Fanuc KAREL source: kt00483.KL

-- PROVISIONAL review KL for V770-1; original PC SHA256 eedee7176f4b0b8d41bb8e5626b35325a9c50e701c9c6c733b56d75d0fa50af2
-- Incomplete behavior may be omitted. Consult companion uncertainty JSON. Do not deploy.
PROGRAM KT00483
%NOLOCKGROUP
VAR
  OUT : BOOLEAN
-- UNRESOLVED_DECL P1 type=000101
-- UNRESOLVED_DECL P2 type=000106
BEGIN
  -- UNRESOLVED_PC offsets 5-20; opcodes 2E,22,32,35
  -- UNRESOLVED_PC offsets 25-53; opcodes 49,49,7E,AC,23
  -- UNRESOLVED_PC offsets 58-62; opcodes 7F
END KT00483
